{attribute 'GeneratedUsingTerminal: ATH2000-0250-0022'}
{attribute addProperty BoxType "ATH2000-0250-0022"}
{attribute addProperty Id "A_0014_ATH2050_5501_0022ATH2050_810F0A2D14"}
{attribute addProperty CRC "2210397789"}
{attribute addProperty Size "14"}
TYPE A_0001_ATH2000_0250_0022_83BFFE5D EXTENDS ATH2000_86175B41 :
STRUCT
	{attribute addProperty Name "A_0014_ATH2050_5501_0022"}
	{attribute addProperty PreviousPort "A_0001(ATH2000-0250-0022) : B"}
	A_0014_ATH2050_5501_0022 : ATH2050_810F0A2D;
END_STRUCT
END_TYPE

(* stored: Version 1.2.0.0, ProductVersion 3.1.4024.9
   DUT A_0001_ATH2000_0250_0022_83BFFE5D: Id {af6fd327-8b36-47f5-98b8-49fba8888227} *)
